FUNCTION GetTick : UDINT
VAR_INPUT
END_VAR
VAR
	getTaskTime : GETTASKTIME;		// allow to get time based value, 
	//w1 : WORD;
	//w2 : WORD; 
END_VAR

getTaskTime();
//w1 := UDINT_TO_WORD(SHR(getTaskTime.timeLoDW, 16));
//w2 := UDINT_TO_WORD(getTaskTime.timeLoDW AND 16#FFFF);
//GetTick := SHL(WORD_TO_UDINT(w2), 16) OR w1;
GetTick := getTaskTime.timeLoDW/10000;

END_FUNCTION

(* stored: Version 1.1.0.1, ProductVersion 3.1.4024.6
   POU GetTick: Id {29921add-6e89-4945-967a-5cd442b28ed3}, SpecialFunc None *)
